// TIA Portal V20 export
// export: Created 2025-12-01T14:57:20.85387Z, ExportSetting None, DisplayName Totally Integrated Automation Portal, DisplayVersion V20 Update 3, DisplayName TIA Portal Openness, DisplayVersion V20 Update 3, DisplayName TIA Portal Version Control Interface, DisplayVersion V20 Update 3, DisplayName STEP 7 Professional, DisplayVersion V20 Update 3, DisplayName STEP 7 Safety, DisplayVersion V20 Update 2, DisplayName WinCC Basic/Comfort/Advanced, DisplayVersion V20 Update 3, DisplayName WinCC Professional, DisplayVersion V20 Update 3, DisplayName WinCC Unified, DisplayVersion V20 Update 3
DATA_BLOCK "DB2111_DB_LinPot1"   // DB2111, F_DB
FAMILY : FPRI0853
VERSION : 0.0
// stored: AutoNumber false, InstanceOfName FB2131_F_Linea_Potencia, InstanceOfType FB
"FB2131_F_Linea_Potencia"
   // VAR_INPUT
   //    NumArmario : Int;
   //    NumLinea : Int;
   //    Desconectar : Bool;
   //    Proteccion : Bool;
   //    Seguridades : Bool;
   //    FEEDBACK : Bool;
   //    ACK_NEC : Bool;
   //    ACK : Bool;
   //    "ACK_ESTA _LINEA" : Bool;
   //    QBAD_FIO : Bool;
   //    FDB_TIME : Time;
   //    TIM_Estabilizacion : Time;
   // END_VAR
   // VAR_OUTPUT
   //    Q : Bool;
   //    ERROR : Bool;
   //    ACK_Next : Bool;
   // END_VAR
   // VAR
   //    F_TON { S7_SetPoint := 'True'} : TON;
   //    F_FDBACK { S7_SetPoint := 'True'} : FDBACK;
   //    F_ESTOP1 { S7_SetPoint := 'True'} : ESTOP1;
   //    Mem_ACK : Bool;
   //    Pos_ACK : Bool;
   // END_VAR
BEGIN
END_DATA_BLOCK
